// TwinCAT 3 PLC project SA_function_generator
// ProgramVersion: 3.1.4023.0
// libraries:
//   Tc2_ControllerToolbox, * (Beckhoff Automation GmbH)
//   Tc2_EtherCAT, * (Beckhoff Automation GmbH)
//   Tc2_Standard, * (Beckhoff Automation GmbH)
//   Tc2_System, * (Beckhoff Automation GmbH)
//   Tc2_Utilities, * (Beckhoff Automation GmbH)
//   Tc3_Module, * (Beckhoff Automation GmbH)
//   VisuSymbols,3.5.10.0,System
// project tree:
//   / GlobalTextList.TcGTLO, PlcTask.TcTTO, Visualization Manager.TcVMO (not stored)
//   POUs/ Action_list.TcTLEO, FB_ClearFault.TcPOU, FB_ReadAlias.TcPOU, FB_ReadNcyl.TcPOU, FB_readtextfile.TcPOU, FB_WritePWM.TcPOU, sig_gen.TcPOU, MAIN.TcPOU
//   VISUs/ Visualization.TcVIS
// real-time tasks:
//   TASK PlcTask: cycle T#1ms, priority 20, ADS port 350
// I/O:
//   DEVICE Device 1 (EtherCAT), AmsNetId 10.10.16.19.2.1
//     Box 1 (m1sa) [m1sa]
// variable links:
//   SA_function_generator/SA_function_generator Instance <-> Device 1 (EtherCAT)/Box 1 (m1sa)
//     PlcTask Inputs/MAIN.err_cal <-> Status process data mapping/err_calibrated
//     PlcTask Inputs/MAIN.err_dongle <-> Status process data mapping/err_dongle
//     PlcTask Inputs/MAIN.err_f_minmax <-> Status process data mapping/err_force_minmax
//     PlcTask Inputs/MAIN.err_f_step <-> Status process data mapping/err_force_step
//     PlcTask Inputs/MAIN.err_ff <-> Status process data mapping/err_follow_error
//     PlcTask Inputs/MAIN.err_locid <-> Status process data mapping/err_locid
//     PlcTask Inputs/MAIN.err_mhb <-> Status process data mapping/err_masterhb
//     PlcTask Inputs/MAIN.err_soc <-> Status process data mapping/err_soc
//     PlcTask Inputs/MAIN.pwm1 <-> Status process data mapping/pwm1
//     PlcTask Inputs/MAIN.pwm2 <-> Status process data mapping/pwm2
//     PlcTask Inputs/MAIN.pwm3 <-> Status process data mapping/pwm3
//     PlcTask Inputs/MAIN.rb_x <-> Status process data mapping/force_rb_X
//     PlcTask Inputs/MAIN.rb_y <-> Status process data mapping/force_rb_Y
//     PlcTask Inputs/MAIN.rb_z <-> Status process data mapping/force_rb_Z
//     PlcTask Inputs/MAIN.spr_x <-> Status process data mapping/force_sp_X
//     PlcTask Inputs/MAIN.spr_y <-> Status process data mapping/force_sp_Y
//     PlcTask Inputs/MAIN.spr_z <-> Status process data mapping/force_sp_Z
//     PlcTask Outputs/MAIN.close_loop <-> Control process data mapping/close_loop
//     PlcTask Outputs/MAIN.enable <-> Control process data mapping/enable
//     PlcTask Outputs/MAIN.msthb <-> Control process data mapping/msthb
//     PlcTask Outputs/MAIN.sp_x <-> Control process data mapping/force_sp_X
//     PlcTask Outputs/MAIN.sp_y <-> Control process data mapping/force_sp_Y
//     PlcTask Outputs/MAIN.sp_z <-> Control process data mapping/force_sp_Z

CONFIGURATION SA_function_generator
    RESOURCE PLC ON TwinCAT3
        TASK PlcTask(INTERVAL := T#1ms, PRIORITY := 20);
        PROGRAM MAIN WITH PlcTask : MAIN;
    END_RESOURCE
END_CONFIGURATION

// ---- POUs/Action_list.TcTLEO
{attribute 'qualified_only'}
{attribute 'strict'}
TYPE Action_list :
(
	idle := 0,
	clear_fault := 1,
	enable_all := 2,
	disable_all :=3,
	read_ncyl :=4,
	read_alias :=5,
	read_gains := 6,
	write_gains := 7,
	read_dongle_singlevalue := 8,
	save_soc_all := 9,
	bump_test := 10,
	function_generator := 11
) := idle;
END_TYPE

// ---- POUs/MAIN.TcPOU

PROGRAM MAIN
VAR
	actions : (idle, clear_all, enable_all, disable_all,read_ncyl,read_alias,read_gains,write_gains,read_file,send_waveform_cmd, send_waveform_pwm);
	slave_pos : UINT := 1001;	
	clearfault : FB_ClearFault;
	readncyl : FB_ReadNcyl;
	readalias : FB_ReadAlias;
	readfile : FB_readtextfile;
	waveform_pwm : FB_WritePWM;
	state : INT := 2;
	step : DWORD :=0;
	bError : BOOL;
	t_index : UINT :=1;
	alias : UDINT;
	ncyl: UINT;
	signal : ARRAY[1..60000] OF REAL;
	db : REAL :=14.0;
	dbi : REAL := 0;
	pwm : REAL := 0.0;
	value : REAL := 0.0;
	
	sdo_address: UINT;
	subIndex: BYTE;
	sNetId_local : T_AmsNetId := '10.10.16.19.2.1';	// Address of this computer 
	
// heartbeat
	msthb AT %Q* : UDINT;
	enable AT %Q* : BOOL;
	close_loop AT %Q* : BOOL;
	sp_x AT %Q* : REAL;
	sp_y AT %Q* : REAL;
	sp_z AT %Q* : REAL;
	rb_x AT %I* : REAL;
	rb_y AT %I* : REAL;
	rb_z AT %I* : REAL;
	spr_x AT %I* : REAL;
	spr_y AT %I* : REAL;
	spr_z AT %I* : REAL;
	pwm1 AT %I* : REAL;
	pwm2 AT %I* : REAL;
	pwm3 AT %I* : REAL;
	
	err_mhb AT %I* : BOOL;
	err_f_minmax AT %I* : BOOL;
	err_f_step AT %I* : BOOL;
	err_cal AT %I* : BOOL;
	err_dongle AT %I* : BOOL;
	err_locid AT %I* : BOOL;
	err_soc AT %I* : BOOL;
	err_ff AT %I* : BOOL; 
END_VAR

// send heartbeat to all SA and EPHS

msthb := msthb + 1;


CASE actions OF
	idle:
		state := 2;
		bError := 0;
		t_index := 1;
		sp_x := 0;
		sp_y := 0;
		sp_z := 0;
		
	enable_all :
		enable := TRUE;
		close_loop := TRUE;
		
	disable_all:
		enable := FALSE;
		close_loop := FALSE;
		
	clear_all:
	clearfault(bExecute := TRUE, slv_addr := slave_pos, state => state, bError=> bError );
	IF state = 0 THEN
		actions := idle;
	END_IF
		
	read_ncyl :
		readncyl(bExecute := TRUE, slv_addr := slave_pos, state => state, bError=> bError, value =>ncyl );
		IF state = 0 THEN
			actions := idle;
		END_IF
		
	read_alias :
		readalias(bExecute := TRUE, slv_addr := slave_pos, state => state, bError=> bError, value =>alias );
		IF state = 0 THEN
			actions := idle;
		END_IF
		
	read_file :
		readfile(bread := TRUE,output=>signal,step=>step);
		IF step = 0 THEN
			actions := idle;
		END_IF	
		
	send_waveform_cmd :
	    sp_x := signal[t_index];
		t_index := t_index+1;
		IF t_index>60000 THEN
			t_index := 1;
		END_IF
	
	send_waveform_pwm:
		waveform_pwm(bExecute := TRUE, slv_addr := slave_pos,value :=  6*signal[t_index], state => state, bError=> bError );
		t_index := t_index+1;
		IF t_index>60000 THEN
			t_index := 1;
		END_IF
END_CASE

END_PROGRAM

// ---- POUs/FB_ClearFault.TcPOU
FUNCTION_BLOCK FB_ClearFault
VAR_INPUT
	bExecute : BOOL := FALSE;
	slv_addr : UINT := 0;
END_VAR
VAR_OUTPUT
	state : INT := 0;
	
	bError : BOOL;
	
END_VAR
VAR
	fbSdoWrite : FB_EcCoESdoWrite;
	nErrID : UDINT :=0;
	sdo_address: UINT := 16#8006;
	subIndex: BYTE := 1;
	value : INT := 1;
END_VAR

//IF MAIN.write_action = TRUE THEN
//	bExecute := TRUE;
//	IF delay_cycle = 10 THEN
//		IF slv_addr < 1182 THEN
//			slv_addr := slv_addr + 1;
//		ELSE
//			slv_addr := 1002;
//		END_IF
//		CASE  slv_addr OF
//			1001,1018,1033,1046,1063,1080,1097,1114,1131,1148,1165:
//			slv_addr := slv_addr+1;
//		END_CASE
//		delay_cycle := 1;
//	ELSE
//		delay_cycle := delay_cycle+1;	
//	END_IF
//ELSE
//	bExecute := FALSE;
//	slv_addr := 1002;
//	index := 1;
//	delay_cycle := 1;
//END_IF

fbSdoWrite(
        sNetId          := MAIN.sNetId_local,
        //nSlaveAddr      := nSlaveAddr,
		nSlaveAddr :=   slv_addr,
        nIndex          := sdo_address,
        nSubIndex       := subIndex,
        pSrcBuf         := ADR(value),
        cbBufLen        := SIZEOF(value),
        bExecute        := bExecute
);
state := 1;
IF NOT fbSdoWrite.bBusy THEN
        bExecute := FALSE;
		//done	:= TRUE;
        IF NOT bError THEN 
                (* write successful *)
                bError := FALSE;
                nErrId := 0;
        ELSE 
                (* write failed *)
                bError := fbSdoWrite.bError;
                nErrId := fbSdoWrite.nErrId;
        END_IF
        fbSdoWrite(bExecute := FALSE);
		state := 0;
END_IF

END_FUNCTION_BLOCK

// ---- POUs/FB_ReadNcyl.TcPOU
FUNCTION_BLOCK FB_ReadNcyl
VAR_INPUT
	bExecute : BOOL := FALSE;
	slv_addr : UINT := 0;
END_VAR
VAR_OUTPUT
	state : INT := 0;
	bError : BOOL;
	value : UINT;
	
END_VAR
VAR
	fbSdoRead : FB_EcCoESdoRead;
	nErrID : UDINT :=0;
	sdo_address: UINT := 16#8005;
	subIndex: BYTE := 5;
	
END_VAR

fbSdoRead(
        sNetId          := MAIN.sNetId_local,
        //nSlaveAddr      := nSlaveAddr,
		nSlaveAddr :=   slv_addr,
        nIndex          := sdo_address,
        nSubIndex       := subIndex,
        pDstBuf         := ADR(value),
        cbBufLen        := SIZEOF(value),
        bExecute        := bExecute
);
state := 1;
IF NOT fbSdoRead.bBusy THEN
        bExecute := FALSE;
		//done	:= TRUE;
        IF NOT bError THEN 
                (* write successful *)
                bError := FALSE;
                nErrId := 0;
        ELSE 
                (* write failed *)
                bError := fbSdoRead.bError;
                nErrId := fbSdoRead.nErrId;
        END_IF
        fbSdoRead(bExecute := FALSE);
		state := 0;
END_IF

END_FUNCTION_BLOCK

// ---- POUs/FB_ReadAlias.TcPOU
FUNCTION_BLOCK FB_ReadAlias
VAR_INPUT
	bExecute : BOOL := FALSE;
	slv_addr : UINT := 0;
END_VAR
VAR_OUTPUT
	state : INT := 0;
	bError : BOOL;
	value : UDINT := 0;
	
END_VAR
VAR
	fbSdoRead : FB_EcCoESdoRead;
	nErrID : UDINT :=0;
	sdo_address: UINT := 16#8008;
	subIndex: BYTE := 1;
	
END_VAR

fbSdoRead(
        sNetId          := MAIN.sNetId_local,
        //nSlaveAddr      := nSlaveAddr,
		nSlaveAddr :=   slv_addr,
        nIndex          := sdo_address,
        nSubIndex       := subIndex,
        pDstBuf         := ADR(value),
        cbBufLen        := SIZEOF(value),
        bExecute        := bExecute
);
state := 1;
IF NOT fbSdoRead.bBusy THEN
        bExecute := FALSE;
		//done	:= TRUE;
        IF NOT bError THEN 
                (* write successful *)
                bError := FALSE;
                nErrId := 0;
        ELSE 
                (* write failed *)
                bError := fbSdoRead.bError;
                nErrId := fbSdoRead.nErrId;
        END_IF
        fbSdoRead(bExecute := FALSE);
		state := 0;
END_IF

END_FUNCTION_BLOCK

// ---- POUs/FB_readtextfile.TcPOU
FUNCTION_BLOCK FB_readtextfile
VAR_INPUT
	bRead : BOOL :=FALSE;
END_VAR
VAR_OUTPUT
	step			: DWORD 	:= 0;
	output : ARRAY[1..60000] OF REAL;
END_VAR
VAR
	//bRead			: BOOL := FALSE;(* Rising edge starts program execution *)
	sNetId			: T_AmsNetId := '10.10.16.19.1.1';	(* TwinCAT system network address *)
	sFileName		: T_MaxString := 'C:\Users\tranka\Documents\TestCellFeb22\sinesweep_TAMU1_0offset_250Hz.csv';(* CSV source file path and name *)
	sCSVLine		: T_MaxString := '';(* Single CSV text line (row, record), we are using string as record buffer (your are able to see read fields)  *)
	sCSVField		: T_MaxString := '';(* Single CSV field value (column, record field) *)
	bBusy			: BOOL;
	bError			: BOOL;
	nErrId			: UDINT;
	nRow	 		: UDINT 	:= 1;(* Row number (record) *)
	nColumn			: UDINT 	:= 0;(* Column number (record field) *)
	hFile			: UINT		:= 0;(* File handle of the source file *)
	
	fbFileOpen		: FB_FileOpen;(* Opens file *)
	fbFileClose		: FB_FileClose;(* Closes file *)
	fbFileGets		: FB_FileGets;(* Reads one record (line) *)
	fbReader		: FB_CSVMemBufferReader;(* Helper function block used to parse CSV data bytes (single record line) *)

	database		: ARRAY[1..60000] OF STRING(100);(* Target PLC database *)
	MAX_CSV_ROWS: UDINT := 60000;
	//MAX_CSV_COLUMNS: UDINT:= 1;
END_VAR

CASE step OF
	0:	(* Wait for rising edge at bRead variable *)
		IF bRead THEN
			bRead 	:= FALSE;
			bBusy 	:= TRUE;
			bError	:= FALSE;
			nErrId	:= 0;
			hFile	:= 0;
			nRow	:= 1;
			//nColumn	:= 0;
			MEMSET( ADR( database ), 0, SIZEOF( database ) );
			step 		:= 1;
		END_IF

	1:	(* Open source file *)
		fbFileOpen(  bExecute := FALSE  );
		fbFileOpen( sNetId := sNetId, sPathName := sFileName, nMode := FOPEN_MODEREAD OR FOPEN_MODETEXT,(* Open file in TEXT mode! *)
					ePath := PATH_GENERIC, bExecute := TRUE );
		step := 2;

	2:(* Wait until open not busy *)
		fbFileOpen( bExecute := FALSE, bError => bError, nErrID => nErrID, hFile => hFile );
		IF NOT fbFileOpen.bBusy THEN
			IF NOT fbFileOpen.bError THEN
				step := 3;
			ELSE(* Error: file not found? *)
				step := 100;
			END_IF
		END_IF

	3:	(* Read single line (record) *)
		fbFileGets( bExecute := FALSE );
		fbFileGets( sNetId := sNetId, hFile := hFile, bExecute := TRUE );
		step := 4;

	4:(* Wait until read not busy *)
		fbFileGets( bExecute := FALSE, bError => bError, nErrID => nErrID, sLine => sCSVLine );
		IF NOT fbFileGets.bBusy THEN
			IF NOT fbFileGets.bError THEN
				IF fbFileGets.bEOF THEN
					step := 10;(* End of file reached => Close source file *)
				ELSE

					(* FB_FileGets returns text line without the CR (carriage return) character.
					We have to restore the CR character (replace the $L character with $R$L characters) *)
					IF RIGHT( sCSVLine, 1 ) = '$L' THEN
						sCSVLine := REPLACE( sCSVLine, '$R$L', 2, LEN( sCSVLine ) );
					END_IF

					step := 5;
				END_IF
			ELSE(* Error *)
				step := 100;
			END_IF
		END_IF

	5:(* Parse single line (record) *)
		fbReader.eCmd := eEnumCmd_First;(* Read first field value *)
		REPEAT
			fbReader( pBuffer := ADR( sCSVLine ), cbBuffer := SIZEOF( sCSVLine ), getValue => sCSVField );
			IF fbReader.bOk THEN
				fbReader.eCmd := eEnumCmd_Next;(* Read next field value *)

				IF ( nRow <= MAX_CSV_ROWS ) THEN
					//IF ( nColumn <= MAX_CSV_COLUMNS ) THEN
						database[nRow] := CSVFIELD_TO_STRING( sCSVField, FALSE );(* TODO: Save or use the field value in your application *)
						output[nRow] := STRING_TO_REAL(database[nRow]);
					//END_IF
				END_IF

				//nColumn := nColumn + 1;(* Increment number of read columns *)
				IF fbReader.bCRLF THEN(* CRLF == TRUE => End of reacord reached *)
					nRow 		:= nRow + 1;(* Increment number of read records *)
					//nColumn 	:= 0;(* Reset number of columns *)
				END_IF

			ELSE(* Error: End of record reached or all fields read *)
				step := 3;(* Try to read next line *)
			END_IF
		UNTIL NOT fbReader.bOk
		END_REPEAT

	10:	(* Close source file *)
		fbFileClose( bExecute := FALSE );
		fbFileClose( sNetId := sNetId, hFile := hFile, bExecute := TRUE );
		step := 11;

	11:(* Wait until close not busy *)
		fbFileClose( bExecute := FALSE, bError => bError, nErrID => nErrID );
		IF ( NOT fbFileClose.bBusy ) THEN
			hFile := 0;
			step := 100;
		END_IF

	100: (* Error or ready step => cleanup *)
		IF ( hFile <> 0 ) THEN
			step := 10; (* Close the source file *)
		ELSE
			bBusy := FALSE;
			step := 0;	(* Ready *)
		END_IF

END_CASE

END_FUNCTION_BLOCK

// ---- POUs/FB_WritePWM.TcPOU
FUNCTION_BLOCK FB_WritePWM
VAR_INPUT
	bExecute : BOOL := FALSE;
	slv_addr : UINT := 0;
	value : REAL := 0.0;
END_VAR
VAR_OUTPUT
	state : INT := 0;
	bError : BOOL;
END_VAR
VAR
	fbSdoWrite : FB_EcCoESdoWrite;
	nErrID : UDINT :=0;
	sdo_address: UINT := 16#8001;
	subIndex: BYTE := 7;
END_VAR

fbSdoWrite(
        sNetId          := MAIN.sNetId_local,
        //nSlaveAddr      := nSlaveAddr,
		nSlaveAddr :=   slv_addr,
        nIndex          := sdo_address,
        nSubIndex       := subIndex,
        pSrcBuf         := ADR(value),
        cbBufLen        := SIZEOF(value),
        bExecute        := bExecute
);
state := 1;
IF NOT fbSdoWrite.bBusy THEN
        bExecute := FALSE;
		//done	:= TRUE;
        IF NOT bError THEN 
                (* write successful *)
                bError := FALSE;
                nErrId := 0;
        ELSE 
                (* write failed *)
                bError := fbSdoWrite.bError;
                nErrId := fbSdoWrite.nErrId;
        END_IF
        fbSdoWrite(bExecute := FALSE);
		state := 0;
END_IF

END_FUNCTION_BLOCK

// ---- POUs/sig_gen.TcPOU
PROGRAM sig_gen
VAR
	FB_sig_gen : FB_CTRL_SIGNAL_GENERATOR;
	sig_gen_params : ST_CTRL_SIGNAL_GENERATOR_PARAMS :=(eSignalType:=1,tTaskCycleTime := T#1MS,tCtrlCycleTime := T#1MS, tCylceDuration := T#2S,tStart := T#0S,fAmplitude:=10,fOffset:=5);
	operating_mode : E_CTRL_MODE;
	manual_auto : INT := 2;
	fManValue : LREAL;
	
	eState    : E_CTRL_STATE;
    eErrorId  : E_CTRL_ERRORCODES;
    bError    : BOOL;
	sig_output : REAL;
	c: INT;
END_VAR

operating_mode := manual_auto;
IF operating_mode = manual_auto THEN
	FB_sig_gen(fManValue:=fManValue, eMode :=operating_mode, stParams:=sig_gen_params,eState=>eState,eErrorId=>eErrorId, bError=>bError, fOut=>sig_output);
	operating_mode := 0;
	c := c+1;
END_IF

END_PROGRAM

// ---- GlobalTextList.TcGTLO
TEXTLIST GlobalTextList
  450 = 'actions'
  46 = 'SA Error bits'
END_TEXTLIST

// ---- VISUs/Visualization.TcVIS
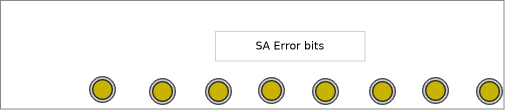
VISUALIZATION Visualization  // 505x110
    Lamp1 (310,73 31x37), variable: MAIN.err_ff, style: Lamp-Lamp1-Yellow
    Lamp1 (256,72 31x37), variable: MAIN.err_f_step, style: Lamp-Lamp1-Yellow
    Lamp1 (203,73 31x37), variable: MAIN.err_f_minmax, style: Lamp-Lamp1-Yellow
    Lamp1 (147,73 31x37), variable: MAIN.err_dongle, style: Lamp-Lamp1-Yellow
    Lamp1 (87,71 31x37), variable: MAIN.err_cal, style: Lamp-Lamp1-Yellow
    Lamp1 (474,73 31x37), variable: MAIN.err_soc, style: Lamp-Lamp1-Yellow
    Lamp1 (420,72 31x37), variable: MAIN.err_mhb, style: Lamp-Lamp1-Yellow
    Lamp1 (367,73 31x37), variable: MAIN.err_locid, style: Lamp-Lamp1-Yellow
    Textfield (215,31 150x30), "SA Error bits"
END_VISUALIZATION
